(* CODESYS project Tintas.project

Project tree, tasks and I/O mapping:
  Device : CODESYS Control Win V3 x64, 3S - Smart Software Solutions GmbH, version 3.5.11.30
    application Application
      libraries: Standard, * (System)
      task MainTask (cyclic, interval t#20ms, priority 1) calls PLC_PRG
      task VISU_TASK (cyclic, interval 100 ms, priority 31) calls VisuElems.Visu_Prg
      program PLC_PRG [LD]
      visualisation Visualization
  libraries: VisuSymbols, 3.5.10.0 (System)
  text list GlobalTextList
*)

// Device/Application/PLC_PRG
PROGRAM PLC_PRG
VAR
	BOMBA1: BOOL;
	LIGA1: BOOL;
	DESLIGA1: BOOL;
	LIGA2: BOOL;
	BOMBA2: BOOL;
	DESLIGA2: BOOL;
	NIVEL_MAXIMO: BOOL;
	MISTURADOR: BOOL;
	VALVULA_VAPOR: BOOL;
	TON1: TON;
	VALVULA_DRENO: BOOL;
	NIVEL_MINIMO: BOOL;
	TON2: TON;
	BOMBA_DRENO: BOOL;
	FLAG1: BOOL;
END_VAR

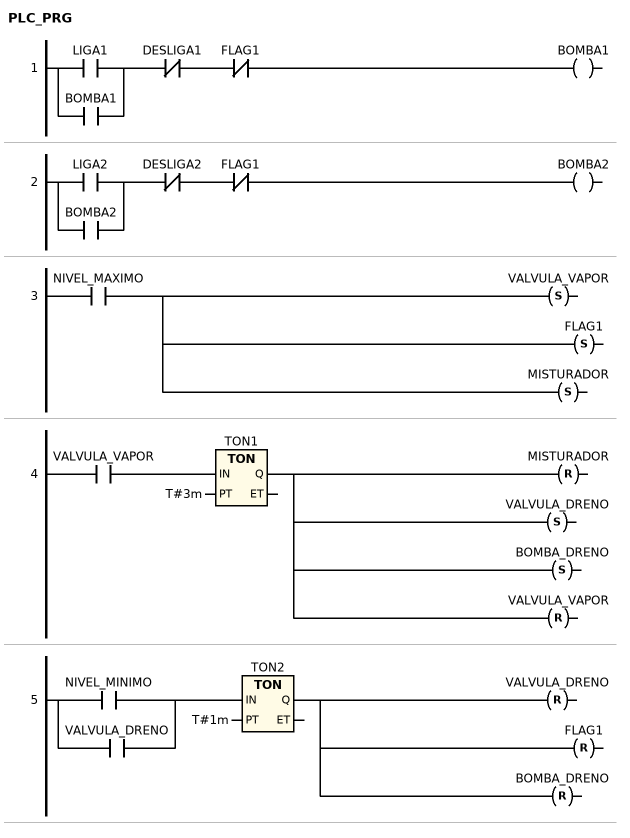
// NETWORK 1
BOMBA1 := (LIGA1 OR BOMBA1) AND NOT DESLIGA1 AND NOT FLAG1;

// NETWORK 2
BOMBA2 := (LIGA2 OR BOMBA2) AND NOT DESLIGA2 AND NOT FLAG1;

// NETWORK 3
VALVULA_VAPOR S= NIVEL_MAXIMO;
FLAG1 S= NIVEL_MAXIMO;
MISTURADOR S= NIVEL_MAXIMO;

// NETWORK 4
TON1(IN := VALVULA_VAPOR, PT := T#3m); // TON
MISTURADOR R= TON1.Q;
VALVULA_DRENO S= TON1.Q;
BOMBA_DRENO S= TON1.Q;
VALVULA_VAPOR R= TON1.Q;

// NETWORK 5
TON2(IN := NIVEL_MINIMO OR VALVULA_DRENO, PT := T#1m); // TON
VALVULA_DRENO R= TON2.Q;
FLAG1 R= TON2.Q;
BOMBA_DRENO R= TON2.Q;

END_PROGRAM

// Device/Application/Visualization
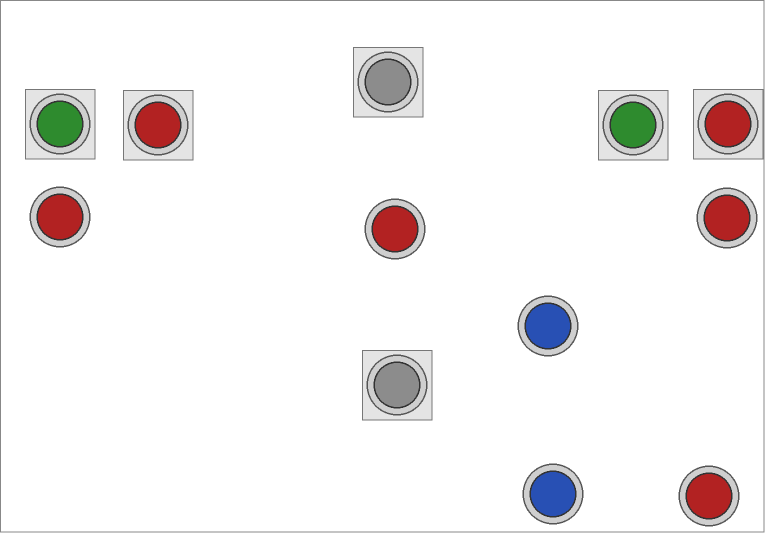
VISUALIZATION Visualization  // 765x533
    Lamp1 (25,182 70x70), variable: PLC_PRG.BOMBA1, style: Lamp-Lamp1-Red
    Lamp1 (692,183 70x70), variable: PLC_PRG.BOMBA2, style: Lamp-Lamp1-Red
    PushSwitch (25,89 70x70), variable: PLC_PRG.LIGA1, behaviour: TAP, style: Switch-PushSwitch-Green
    PushSwitch (123,90 70x70), variable: PLC_PRG.DESLIGA1, behaviour: TAP, style: Switch-PushSwitch-Red
    PushSwitch (598,90 70x70), variable: PLC_PRG.LIGA2, behaviour: TAP, style: Switch-PushSwitch-Green
    PushSwitch (693,89 70x70), variable: PLC_PRG.DESLIGA2, behaviour: TAP, style: Switch-PushSwitch-Red
    Lamp1 (360,194 70x70), variable: PLC_PRG.MISTURADOR, style: Lamp-Lamp1-Red
    Lamp1 (513,291 70x70), variable: PLC_PRG.VALVULA_VAPOR, style: Lamp-Lamp1-Blue
    Lamp1 (518,459 70x70), variable: PLC_PRG.VALVULA_DRENO, style: Lamp-Lamp1-Blue
    Lamp1 (674,461 70x70), variable: PLC_PRG.BOMBA_DRENO, style: Lamp-Lamp1-Red
    PushSwitch (353,47 70x70), variable: PLC_PRG.NIVEL_MAXIMO, behaviour: TAP, style: Switch-PushSwitch-Gray
    PushSwitch (362,350 70x70), variable: PLC_PRG.NIVEL_MINIMO, behaviour: TAP, style: Switch-PushSwitch-Gray
END_VISUALIZATION
